// TIA Portal V19 export
TYPE "stItemListRecipe"
   STRUCT
      RecipeName { ExternalAccessible := 'False'; ExternalVisible := 'False'; ExternalWritable := 'False'} : String[30];
      RecipeIndex { ExternalAccessible := 'False'; ExternalVisible := 'False'; ExternalWritable := 'False'} : USInt;
   END_STRUCT;
END_TYPE
